FUNCTION_BLOCK VVI_LRI
  (* Standard: 61499-2 *)
  (* Version 0.1, 2014-00-18, Canto-Air, CANTO-AIR-PC *)
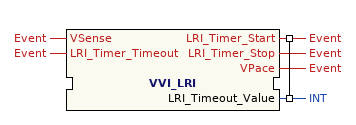
  EVENT_INPUT
    VSense;
    LRI_Timer_Timeout;
  END_EVENT
  EVENT_OUTPUT
    LRI_Timer_Start WITH LRI_Timeout_Value;
    LRI_Timer_Stop;
    VPace;
  END_EVENT
  VAR_OUTPUT
    LRI_Timeout_Value : INT;
  END_VAR
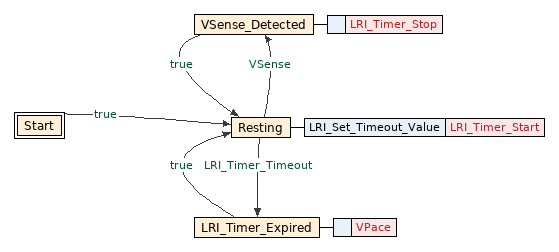
  EC_STATES
    Start;
    Resting : LRI_Set_Timeout_Value -> LRI_Timer_Start;
    LRI_Timer_Expired : -> VPace;
    VSense_Detected : -> LRI_Timer_Stop;
  END_STATES
  EC_TRANSITIONS
    Start TO Resting := true;
    Resting TO VSense_Detected := VSense;
    Resting TO LRI_Timer_Expired := LRI_Timer_Timeout;
    LRI_Timer_Expired TO Resting := true;
    VSense_Detected TO Resting := true;
  END_TRANSITIONS
  ALGORITHM LRI_Set_Timeout_Value IN ST:
LRI_Timeout_Value := 800;
  END_ALGORITHM
END_FUNCTION_BLOCK
